PROGRAM MAIN
VAR
	bVar : BOOL;
	myExternalDB : ExternalDB;
	bInit : BOOL := TRUE;
	bCheck : BOOL;
	udiRes : VUM_ReturnValues;
END_VAR

IF bInit THEN
	myExternalDB();
	VisuUserManagement.g_VisuUserMgmt.RegisterExternalUserDatabaseProvider(myExternalDB);
	bInit := FALSE;
END_IF

END_PROGRAM

(* stored: Version 1.1.0.1, ProductVersion 3.1.4020.2
   POU MAIN: Id {8aae1379-95ca-4993-8d5b-39e2c9872fce}, SpecialFunc None *)
